INTERFACE IACMethod EXTENDS IACObject

PROPERTY IsValid : BOOL
GET
END_GET
END_PROPERTY

END_INTERFACE

(* stored: Version 1.1.0.1, ProductVersion 3.1.4020.12
   Itf IACMethod: Id {749bf654-4a4b-4f5a-bd03-9adffb4ebd84}
   Property IsValid: Id {39d7fa7a-776a-4cf8-952e-8d495cf1d333}
   Get Get: Id {795dc368-6ca7-4904-b5ff-6159f7975509} *)
